(* IEC 61131-3 sources: nvidia-ai-factory-controls/libraries/AIFactory_Communication/POUs/Publishers, 4 files *)

(* ---- FB_Publisher_BACnet.fb ---- *)
(* =============================================================================
    FB_Publisher_BACnet — BACnet/IP Server Publisher
    Common Library | NVIDIA AI Factory Controls
   =============================================================================

   PURPOSE:
     Implements I_DataPublisher by exposing data as BACnet objects.
     External BMS (Building Management Systems) read these values
     using standard BACnet/IP polling (Who-Is/I-Am, ReadProperty).

   USE CASE:
     • Integration with Schneider EcoStruxure, Siemens Desigo, Honeywell
     • Exposing cooling data to facility BMS
     • HVAC coordination (free cooling, heat recovery)
     • Energy metering to campus-level BMS
     • Compliance with building automation standards

   BACnet OBJECT MAPPING:
     Each data point maps to a BACnet object:
       • Analog Value (AV) — for REAL process values (temp, flow, power)
       • Binary Value (BV) — for BOOL status/alarms
       • Analog Input (AI) — for read-only sensor values
       • Multi-State Value (MSV) — for enumerations (states, modes)

   OBJECT NUMBERING:
     AV 1-99:     Cooling system (temps, flows, speeds)
     AV 100-199:  Power system (voltage, PUE, energy)
     AV 200-299:  Environment (temp, humidity, dew point)
     BV 1-99:     Alarms (active flags)
     BV 100-199:  Status (running, healthy, etc.)

   REQUIRES:
     CODESYS BACnet/IP Server device in project tree.
     Or: External BACnet gateway translating from OPC UA.

   THREAD SAFETY:
     BACnet server reads from a value table asynchronously.
     This FB writes to the table in Communication_Task.
     BACnet stack handles its own threading internally.
   ============================================================================= *)

(* ═══════════════════════════════════════════════════════════════════════════════
   DECLARATION
   ═══════════════════════════════════════════════════════════════════════════════ *)

FUNCTION_BLOCK FB_Publisher_BACnet IMPLEMENTS I_DataPublisher
VAR_INPUT
    (* --- Configuration --- *)
    nDeviceInstance       : UDINT := 100001; (* BACnet device instance number *)
    sDeviceName          : STRING(64) := 'AI-Factory-Cooling-IPC02';
    nBaseAV              : UINT := 1;        (* Starting Analog Value object number *)
    nBaseBV              : UINT := 1;        (* Starting Binary Value object number *)
END_VAR

VAR
    _bConnected          : BOOL := TRUE;     (* BACnet server always "running" *)
    _nPublishCount       : UDINT;
    _bBatchMode          : BOOL;

    (* --- Object Value Tables --- *)
    (* These arrays are exposed to the BACnet server device.
       In CODESYS: map these to BACnet AV/BV objects in device config. *)
    _afAnalogValues      : ARRAY[1..300] OF REAL;   (* AV present values *)
    _abBinaryValues      : ARRAY[1..200] OF BOOL;   (* BV present values *)
    _anAnalogStatus      : ARRAY[1..300] OF USINT;  (* BACnet reliability enum *)

    (* --- Object-to-NodePath Mapping --- *)
    _asAV_Map            : ARRAY[1..300] OF STRING(128);  (* AV# → node path *)
    _asBV_Map            : ARRAY[1..200] OF STRING(128);  (* BV# → node path *)
    _nMappedAV           : UINT;
    _nMappedBV           : UINT;

    (* --- Priority Array Support --- *)
    (* BACnet priority arrays (1-16) for commandable objects.
       Priority 1 = Manual Override, 8 = Normal, 16 = Default *)
    _nWritePriority      : USINT := 8;      (* Default write at priority 8 *)
END_VAR

(* ═══════════════════════════════════════════════════════════════════════════════
   IMPLEMENTATION
   ═══════════════════════════════════════════════════════════════════════════════ *)

(* BACnet server is passive — no cyclic processing needed.
   External BMS polls ReadProperty requests; CODESYS BACnet stack
   reads from _afAnalogValues / _abBinaryValues arrays directly.

   M_PublishFloat writes to the appropriate AV index.
   M_PublishBool writes to the appropriate BV index. *)

(* ---- FB_Publisher_Modbus.fb ---- *)
(* =============================================================================
    FB_Publisher_Modbus — Modbus TCP Slave (Server) Publisher
    Common Library | NVIDIA AI Factory Controls
   =============================================================================

   PURPOSE:
     Implements I_DataPublisher by mapping data points to Modbus holding
     registers. External SCADA/HMI systems can read values via standard
     Modbus TCP polling.

   USE CASE:
     • Legacy SCADA integration (Wonderware, iFIX, Ignition)
     • BMS (Building Management System) integration
     • Third-party monitoring tools
     • Simple HMI panels with Modbus-only capability

   REGISTER MAPPING:
     Each data point is assigned a Modbus register address.
     REAL values occupy 2 registers (32-bit float, IEEE 754).
     BOOL values occupy 1 coil or discrete input.

     Default mapping (configurable):
       Registers 0-99:    System status (power, PUE, etc.)
       Registers 100-299: Cooling data (temps, flows, pressures)
       Registers 300-399: Environment data (temp, humidity)
       Registers 400-499: Safety status
       Registers 500-999: Reserved

   REQUIRES:
     CODESYS Modbus TCP Slave device in the project.
     Register mapping configured in device settings.

   THREAD SAFETY:
     CODESYS Modbus slave reads from a memory-mapped register array.
     This FB writes to that array in Communication_Task.
     The Modbus slave reads asynchronously (driven by external polling).
     REAL values (2 registers) must be written atomically — this FB
     writes both registers in sequence within one scan, and CODESYS
     Modbus driver handles the consistency.
   ============================================================================= *)

(* ═══════════════════════════════════════════════════════════════════════════════
   DECLARATION
   ═══════════════════════════════════════════════════════════════════════════════ *)

FUNCTION_BLOCK FB_Publisher_Modbus IMPLEMENTS I_DataPublisher
VAR_INPUT
    (* --- Configuration --- *)
    nBaseRegister        : UINT := 0;       (* Starting register address *)
    nMaxRegisters        : UINT := 1000;    (* Total register space available *)
    nSlaveID             : USINT := 1;      (* Modbus slave/unit ID *)
END_VAR

VAR
    _bConnected          : BOOL := TRUE;    (* Always "connected" — passive slave *)
    _nPublishCount       : UDINT;
    _nNextRegister       : UINT;            (* Next available register for mapping *)

    (* Register-to-NodePath mapping table *)
    _asRegisterMap       : ARRAY[0..499] OF STRING(128);  (* Register → node path *)
    _nMappedCount        : UINT;

    (* Holding register array (exposed to Modbus slave device) *)
    (* In real project: this would be the Modbus slave's register array *)
    _anHoldingRegisters  : ARRAY[0..999] OF WORD;

    _bBatchMode          : BOOL;
END_VAR

(* ═══════════════════════════════════════════════════════════════════════════════
   IMPLEMENTATION
   ═══════════════════════════════════════════════════════════════════════════════ *)

(* Modbus slave is passive — no cyclic processing needed.
   Register array is updated by M_PublishFloat and read by Modbus driver. *)

(* ---- FB_Publisher_MQTT.fb ---- *)
(* =============================================================================
    FB_Publisher_MQTT — MQTT Direct Publisher (Sparkplug B or Plain)
    Common Library | NVIDIA AI Factory Controls
   =============================================================================

   PURPOSE:
     Implements I_DataPublisher using CODESYS MQTT client library.
     Publishes data directly from the PLC to an MQTT broker without
     needing the edge gateway Python bridge.

   USE CASE:
     • Small deployments without edge server
     • Direct-to-cloud publishing (Azure IoT Hub, AWS IoT Core)
     • Redundant path alongside OPC UA
     • Low-latency alarm notification

   PROTOCOLS SUPPORTED:
     • Plain MQTT 3.1.1 / 5.0 (JSON payload)
     • MQTT with Sparkplug B encoding (if library available)

   REQUIRES:
     CODESYS library: IoT_MQTT (CODESYS IoT Libraries Toolkit)
     OR: IoDrvMQTTClient (built-in since CODESYS 3.5 SP17)

   TOPIC STRUCTURE:
     Plain:     {prefix}/{nodePath}    → payload: {"v": 35.2, "q": 0, "t": 1234}
     Sparkplug: spBv1.0/{group}/DDATA/{edge}/{device}

   THREAD SAFETY:
     MQTT client runs in this FB's task context (Communication_Task).
     Publish calls are synchronous (buffered internally by MQTT lib).
     Batch mode collects metrics into one MQTT message for efficiency.
   ============================================================================= *)

(* ═══════════════════════════════════════════════════════════════════════════════
   DECLARATION
   ═══════════════════════════════════════════════════════════════════════════════ *)

FUNCTION_BLOCK FB_Publisher_MQTT IMPLEMENTS I_DataPublisher
VAR_INPUT
    (* --- Broker Configuration --- *)
    sBrokerURL           : STRING(128) := 'tcp://192.168.200.10:1883';
    sClientID            : STRING(64) := 'IPC-02-MQTT';
    sUsername            : STRING(64) := '';
    sPassword            : STRING(64) := '';
    bUseTLS              : BOOL := FALSE;

    (* --- Topic Configuration --- *)
    sTopicPrefix         : STRING(64) := 'aifactory/cooling';
    bUseSparkplug        : BOOL := FALSE;
    sSparkplugGroup      : STRING(32) := 'AIFactory';
    sSparkplugEdgeNode   : STRING(32) := 'IPC_Cooling';

    (* --- QoS --- *)
    nQoS                 : USINT := 0;      (* 0=at-most-once, 1=at-least-once *)
    bRetain              : BOOL := FALSE;
END_VAR

VAR
    _bConnected          : BOOL;
    _nPublishCount       : UDINT;
    _nErrorCount         : UDINT;
    _bBatchMode          : BOOL;

    (* Batch buffer: accumulate metrics then send as one message *)
    _sBatchPayload       : STRING(4096);
    _nBatchItemCount     : UINT;

    (* Connection management *)
    _bConnectRequested   : BOOL;
    _tonReconnect        : TON;
    _tReconnectInterval  : TIME := T#5S;

    (* MQTT client instance (from CODESYS IoT library) *)
    (* _fbMqttClient     : MQTT.MQTTClient;  -- uncomment when library added *)
END_VAR

(* ═══════════════════════════════════════════════════════════════════════════════
   IMPLEMENTATION
   ═══════════════════════════════════════════════════════════════════════════════ *)

(* Connection state machine would run here.
   For now, this is the structural placeholder.
   Actual MQTT library calls added when IoT_MQTT library is imported. *)

(* Auto-reconnect logic *)
IF _bConnectRequested AND NOT _bConnected THEN
    _tonReconnect(IN := TRUE, PT := _tReconnectInterval);
    IF _tonReconnect.Q THEN
        _tonReconnect(IN := FALSE);
        (* Attempt reconnect *)
        (* _fbMqttClient.Connect(...); *)
    END_IF
END_IF

(* ---- FB_Publisher_OPCUA.fb ---- *)
(* =============================================================================
    FB_Publisher_OPCUA — OPC UA Symbol Server Publisher
    Common Library | NVIDIA AI Factory Controls
   =============================================================================

   PURPOSE:
     Implements I_DataPublisher using CODESYS built-in OPC UA server.
     Exposes data points as OPC UA nodes in a hierarchical namespace.

   HOW IT WORKS:
     CODESYS OPC UA server automatically exposes variables marked with
     {attribute 'symbol' := 'readwrite'}. This FB maintains a GVL of
     publishable variables that the OPC UA server reads directly.

     For dynamic publishing (data points registered at runtime), this FB
     writes values to a pre-allocated array in GVL_OPCUA_Publish which
     is exposed to OPC UA via symbol configuration.

   CONFIGURATION:
     The CODESYS OPC UA Server device must be added to the project with:
       • Symbol configuration including GVL_OPCUA_Publish
       • Security: Sign & Encrypt with X.509 certificates
       • Endpoint: opc.tcp://{ip}:4840

   ALTERNATIVE APPROACH:
     For fully dynamic node creation, use CmpOPCUAServer library with
     IecVarAccess. This FB uses the simpler GVL-based approach.
   ============================================================================= *)

(* ═══════════════════════════════════════════════════════════════════════════════
   DECLARATION
   ═══════════════════════════════════════════════════════════════════════════════ *)

FUNCTION_BLOCK FB_Publisher_OPCUA IMPLEMENTS I_DataPublisher
VAR
    _bConnected          : BOOL;
    _nPublishCount       : UDINT;
    _nErrorCount         : UDINT;
    _bBatchMode          : BOOL;
END_VAR

(* ═══════════════════════════════════════════════════════════════════════════════
   IMPLEMENTATION
   ═══════════════════════════════════════════════════════════════════════════════ *)

(* OPC UA server is always running as part of CODESYS runtime.
   No cyclic processing needed — values are read directly from GVL by server. *)
